// TIA Portal project "ISA_P4b" (V16)

(* hardware
DEVICE "S7-1200 station_1"  S7-1200 Station
   slot 0: "Rack_0"  S7-1200 Rack  Rack  V1.0
   slot 1: "PLC_1"  CPU 1215C DC/DC/DC  6ES7 215-1AG40-0XB0  V4.4
DEVICE "PC-System_1"  SIMATIC PC station
   slot 0: "Estación PC SIMATIC"  Rail  SIMATIC PC-Station  V1.0
      slot 125: "Stationmanager"  Station_Manager  V6.0.4
   slot 1: "HMI_RT_1"  WinCC RT Advanced  6AV2 104-0xxxx-xxxx  16.0.0.0
      slot 33792: "Interfaz del equipo"  Host interface
   slot 2: "IE general_1"  IE General  IE_CP  V8.2.0
*)

// ===== PLC "PLC_1"  CPU 1215C DC/DC/DC =====

VAR_GLOBAL   // PLC tag table "Tabla de variables estándar"
   "Tag_1" AT %Q0.0 : Bool;
   "Sync" AT %I0.3 : Bool;
   "Gate" AT %I1.0 : Bool;
   "System_Byte" AT %MB1 : Byte;
   "FirstScan" AT %M1.0 : Bool;
   "DiagStatusUpdate" AT %M1.1 : Bool;
   "AlwaysTRUE" AT %M1.2 : Bool;
   "AlwaysFALSE" AT %M1.3 : Bool;
   "Encoder" AT %ID1000 : DWord;
END_VAR

DATA_BLOCK "Variables"   // DB1
{ S7_Optimized_Access := 'TRUE' }
VERSION : 0.1
   VAR
      resolution : Int;
      diameter : Int;
      distance : Int;
      En_HSC : Bool;
      En_Sync : Bool;
      En_Reference1 : Bool;
      En_CV : Bool;
      En_SV : Bool;
      CV : Int;
      SV : Int;
      Reference1 : Int;
   END_VAR
BEGIN
END_DATA_BLOCK

DATA_BLOCK "Data_block_1"   // DB3
{ S7_Optimized_Access := 'TRUE' }
VERSION : 0.1
   VAR
      MyHSC : HSC_Count;
   END_VAR
BEGIN
   MyHSC.NewReference2 := 0;
   MyHSC.EnHSC := 1;
   MyHSC.EnCapture := false;
   MyHSC.EnSync := 1;
   MyHSC.EnReference1 := 0;
   MyHSC.NewReference1 := 0;
   MyHSC.EnCV := 0;
   MyHSC.EnSV := 1;
   MyHSC.NewStartValue := 30;
END_DATA_BLOCK

ORGANIZATION_BLOCK "Encoder Control"   // OB1, LAD, ProgramCycle
TITLE = "Main Program Sweep (Cycle)"
{ S7_Optimized_Access := 'TRUE' }
VERSION : 0.1
   VAR_INPUT
      Initial_Call : Bool;   // Initial call of this OB
      Remanence : Bool;   // =True, if remanent data are available
   END_VAR
BEGIN

REGION Network 1
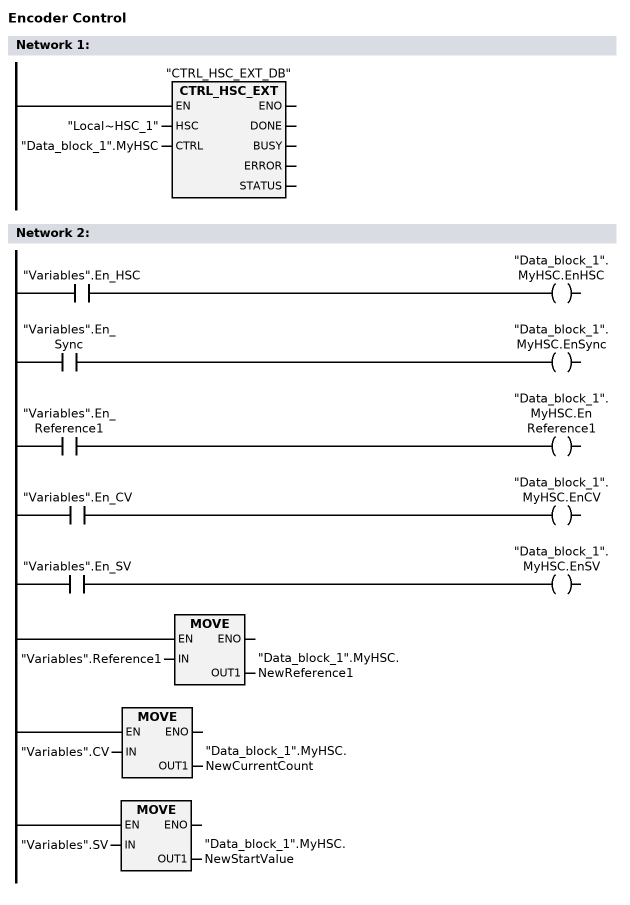
   "CTRL_HSC_EXT_DB"(HSC := "Local~HSC_1", CTRL := "Data_block_1".MyHSC);   // CTRL_HSC_EXT
END_REGION

REGION Network 2
   RUNG wire#powerrail
      Contact( "Variables".En_HSC )
      Coil( "Data_block_1".MyHSC.EnHSC )
   END_RUNG
   RUNG wire#powerrail
      Contact( "Variables".En_Sync )
      Coil( "Data_block_1".MyHSC.EnSync )
   END_RUNG
   RUNG wire#powerrail
      Contact( "Variables".En_Reference1 )
      Coil( "Data_block_1".MyHSC.EnReference1 )
   END_RUNG
   RUNG wire#powerrail
      Contact( "Variables".En_CV )
      Coil( "Data_block_1".MyHSC.EnCV )
   END_RUNG
   RUNG wire#powerrail
      Contact( "Variables".En_SV )
      Coil( "Data_block_1".MyHSC.EnSV )
   END_RUNG
   RUNG wire#powerrail
      Move(in := "Variables".Reference1, out1 => "Data_block_1".MyHSC.NewReference1)
   END_RUNG
   RUNG wire#powerrail
      Move(in := "Variables".CV, out1 => "Data_block_1".MyHSC.NewCurrentCount)
   END_RUNG
   RUNG wire#powerrail
      Move(in := "Variables".SV, out1 => "Data_block_1".MyHSC.NewStartValue)
   END_RUNG
   // the same network as SCL:
   "Data_block_1".MyHSC.EnHSC := "Variables".En_HSC;
   "Data_block_1".MyHSC.EnSync := "Variables".En_Sync;
   "Data_block_1".MyHSC.EnReference1 := "Variables".En_Reference1;
   "Data_block_1".MyHSC.EnCV := "Variables".En_CV;
   "Data_block_1".MyHSC.EnSV := "Variables".En_SV;
   "Data_block_1".MyHSC.NewReference1 := "Variables".Reference1;
   "Data_block_1".MyHSC.NewCurrentCount := "Variables".CV;
   "Data_block_1".MyHSC.NewStartValue := "Variables".SV;
END_REGION
END_ORGANIZATION_BLOCK

ORGANIZATION_BLOCK "Hardware interrupt"   // OB40, LAD, HWProcessInterrupt
{ S7_Optimized_Access := 'TRUE' }
VERSION : 0.1
   VAR_INPUT
      LADDR : Hw_Io;   // Hardware identifier
      USI : Word;   // User structure identifier
      IChannel : USInt;   // Interrupt channel number
      EventType : Byte;   // EventType
   END_VAR
BEGIN

REGION Network 1
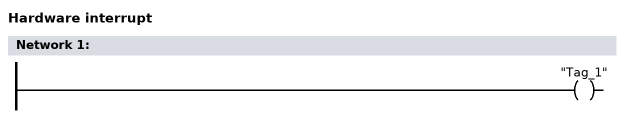
   RUNG wire#powerrail
      Coil( "Tag_1" )
   END_RUNG
   // the same network as SCL:
   "Tag_1" := TRUE;
END_REGION
END_ORGANIZATION_BLOCK

ORGANIZATION_BLOCK "Cálculos"   // OB123, LAD, ProgramCycle
TITLE = "Main Program Sweep (Cycle)"
{ S7_Optimized_Access := 'TRUE' }
VERSION : 0.1
   VAR_INPUT
      Initial_Call : Bool;   // Initial call of this OB
      Remanence : Bool;   // =True, if remanent data are available
   END_VAR
   VAR CONSTANT
      pi : Real := 3.14169;
   END_VAR
BEGIN

REGION Network 1 (SCL)
   "Variables".distance := ("Encoder" * "Variables".diameter * #pi) / "Variables".resolution;
END_REGION
END_ORGANIZATION_BLOCK

(* ===== HMI "HMI_RT_1" =====
system functions are stored by id; their names below are inferred from use
connection "HMI_Conexión_1": ETHERNET, S7_1200_OMS

HMI tags "Tabla de variables estándar"
   "Variables_distance" : Int = PLC Variables.distance, 1 s
   "Variables_Resolution" : Int = PLC Variables.resolution, 1 s
   "Variables_Diámeter" : Int = PLC Variables.diameter, 1 s
   "Tag_1" : Bool = PLC Tag_1 AT %Q0.0, 1 s
   "Encoder" : DWord = PLC Encoder AT %ID1000, 1 s
   "Variables_En_HSC" : Bool = PLC Variables.En_HSC, 1 s
   "Variables_En_Sync" : Bool = PLC Variables.En_Sync, 1 s
   "Variables_En_Reference1" : Bool = PLC Variables.En_Reference1, 1 s
   "Variables_Reference1" : Int = PLC Variables.Reference1, 1 s
   "Variables_CV" : Int = PLC Variables.CV, 1 s
   "Variables_En_CV" : Bool = PLC Variables.En_CV, 1 s
   "Variables_En_SV" : Bool = PLC Variables.En_SV, 1 s
   "Variables_SV" : Int = PLC Variables.SV, 1 s

screen "Imagen_1" 800x600
   IOField "Campo ES_1" at 342,237 size 96x32; FormatPattern s99999
      ProcessValue <- "Variables_distance"
   IOField "Campo ES_2" at 164,143 size 96x32; FormatPattern 99999
      ProcessValue <- "Variables_Resolution"
   IOField "Campo ES_3" at 519,143 size 96x32; FormatPattern 99999
      ProcessValue <- "Variables_Diámeter"
   TextField "Campo de texto_1" at 290,206 size 196x22; Text 'distancia recorrida (mm):'
   TextField "Campo de texto_2" at 148,108 size 130x22; Text 'Resolución (ppr)'
   TextField "Campo de texto_3" at 508,108 size 118x22; Text 'Diámetro (mm)'
   Button "Botón_1" at 341,447 size 96x32; TextOff 'off'
      on Press: ResetBit("Tag_1")
   TextField "Campo de texto_4" at 360,317 size 58x22; Text 'pulsos:'
   IOField "Campo ES_4" at 323,350 size 143x32; FormatPattern 9999999999
      ProcessValue <- "Encoder"
   Switch "Interruptor_1" at 565,327 size 120x57; CaptionText 'EnHSC'; TextOff 'OFF'; TextOn 'ON'
      ProcessValue <- "Variables_En_HSC"
   Switch "Interruptor_2" at 565,414 size 120x57; TextOn 'ON'; CaptionText 'EnSync'; TextOff 'OFF'
      ProcessValue <- "Variables_En_Sync"
   Switch "Interruptor_3" at 53,235 size 95x57; TextOn 'ON'; CaptionText 'EnReference1'; TextOff 'OFF'
      ProcessValue <- "Variables_En_Reference1"
   IOField "Campo ES_5" at 158,255 size 96x32; FormatPattern 99999
      ProcessValue <- "Variables_Reference1"
   Switch "Interruptor_4" at 53,332 size 95x57; TextOn 'ON'; CaptionText 'EnCV'; TextOff 'OFF'
      ProcessValue <- "Variables_En_CV"
   IOField "Campo ES_6" at 158,352 size 96x32; FormatPattern 99999
      ProcessValue <- "Variables_CV"
   Switch "Interruptor_5" at 53,429 size 95x57; TextOn 'ON'; CaptionText 'EnSV'; TextOff 'OFF'
      ProcessValue <- "Variables_En_SV"
   IOField "Campo ES_7" at 158,449 size 96x32; FormatPattern 99999
      ProcessValue <- "Variables_SV"
*)